(* This function use for BurnerControlEcoFlam have Reset by Digital output.
*)
FUNCTION_BLOCK FB_BurnerControlEcoFlamV2 EXTENDS FB_BurnerControlEcoFlam IMPLEMENTS I_BurnerControlEcoFlamV2
VAR
	poReset : FB_DigitalOutput;
	tonReset : TON;
	timeReset : TIME := T#1.5s;
END_VAR

tonReset(
	in := eState=ECOFLAM_RESET,
	PT := timeReset
);
poReset();
poReset.Out := tonReset.IN;
SUPER^();

METHOD PROTECTED MS_Reset : BOOL
piFireSussess.MR_Reset();
bInit 		:= FALSE;
bAbort		:= FALSE;
bIgnition 	:= FALSE;
bStop 		:= FALSE;
IF NOT piFireSussess.ErrorTimedout// for sure least than TimeReset.
	AND tonReset.Q
THEN
	eState := ECOFLAM_RESET_DONE;
END_IF
END_METHOD

PROPERTY Ref_poReset : Reference to FB_DigitalOutput
GET
Ref_poReset ref= poReset;
END_GET
END_PROPERTY

END_FUNCTION_BLOCK

(* stored: Version 1.1.0.1, ProductVersion 3.1.4024.12
   POU FB_BurnerControlEcoFlamV2: Id {890a56d1-1ac8-4d8d-bc91-d02dd763dd8f}, SpecialFunc None
   Folder Internal: Id {bd4dc108-7c01-4c06-855a-5c2e03d60714}
   Method MS_Reset: Id {1073984c-af6c-466e-a7a3-8ad219bb6330}
   Property Ref_poReset: Id {19a4886f-ceaa-4baa-af92-8ae8e5948c09}
   Get Get: Id {837e7930-98a4-4da2-afea-30550f6a972f} *)
